{attribute addProperty BoxType "EPP1518-0002-0016"}
{attribute addProperty Id "InputAT %I*ARRAY[0 ..7] OF BOOL6480"}
{attribute addProperty CRC "1701588874"}
{attribute addProperty SizeInBites "64"}
{attribute addProperty SizeInBytes "8"}
TYPE DIG_Inputs_E017EA69 :
STRUCT
	{attribute addProperty Name "Input"}
	Input AT %I* : ARRAY[0 ..7] OF BOOL;
END_STRUCT
END_TYPE

(* stored: Version 1.2.0.0, ProductVersion 3.1.4024.9
   DUT DIG_Inputs_E017EA69: Id {7a2393ac-c70a-4a64-aaf0-1a04eae1dadc} *)
